// Setpoints for the temperature monitors
TYPE ST_TemperatureMonitorSetpoints :
STRUCT
	{attribute 'pytmc' := '
		pv: MAX_TEMP
		io: io
		field: EGU C
	'}
	fMaxTemperature : LREAL; // Maximum temperature in Celsius allowed before triggering error
END_STRUCT
END_TYPE

(* stored: Version 1.1.0.1, ProductVersion 3.1.4024.6
   DUT ST_TemperatureMonitorSetpoints: Id {15eb5ded-fd00-4e69-b770-6bc69f554886} *)
